RESOURCE_TYPE topMANY
  (* Standard: 61499-2 *)
  (* Version 0.1, 2017-00-14, Hammond, HAMMONDSDESKTOP *)
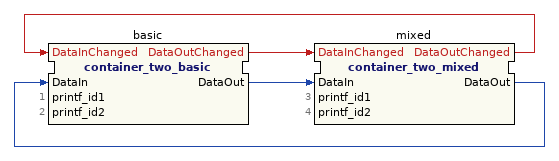
  FBS
    basic : container_two_basic(printf_id1 := 1, printf_id2 := 2);
    mixed : container_two_mixed(printf_id1 := 3, printf_id2 := 4);
  END_FBS
  EVENT_CONNECTIONS
    basic.DataOutChanged TO mixed.DataInChanged;
    mixed.DataOutChanged TO basic.DataInChanged;
  END_CONNECTIONS
  DATA_CONNECTIONS
    basic.DataOut TO mixed.DataIn;
    mixed.DataOut TO basic.DataIn;
  END_CONNECTIONS
END_RESOURCE_TYPE
